Universal Robots PolyScope program: ruch1MS.urp

Program ruch1MS (installation=default directory=/programs/usbdisk createdIn=3.15.8.106339 lastSavedIn=3.15.8.106339 robotSerialNumber=2020330428)
Calibrated DH parameters: a=[0.000029, -0.241913, -0.128453, -0.000049, -0.000012, 0]; d=[0.151842, -4.082088, 33.504745, -29.309875, 0.08529, 0.082285]; alpha=[1.571059, -0.006644, 0.005794, 1.571984, -1.571997, 0]; deltaTheta=[-0.000032, 0.111537, 0.813391, -0.924919, 0.000036, 0.000016]
Robot Program (runOnlyOnce=false)
  MoveJ speed 50 deg/s, acceleration 100 deg/s^2 (useActiveTCP=true)
    Waypoint Punkt_orienta_1: TCP in base x=-541.111 y=-270.483 z=152.712 mm, rx=1.2043 ry=1.2088 rz=-1.2077 rad; joints [-0.004, 0, 0.003, -90, 0, 0] deg; flange x=-541.395 y=-195.484 z=152.496 mm, rx=1.2043 ry=1.2088 rz=-1.2077 rad
    Waypoint Punkt_orienta_3: TCP in base x=541.129 y=-270.562 z=150.788 mm, rx=1.2088 ry=-1.2137 rz=1.2047 rad; joints [-0.001, -180, -0.002, -90.001, 0.004, 0.005] deg; flange x=541.424 y=-195.563 z=151.05 mm, rx=1.2088 ry=-1.2137 rz=1.2047 rad
